FUNCTION_BLOCK Starting IMPLEMENTS ITF_PackMLState
VAR
	_MyContext : REFERENCE TO SomeMachine;
END_VAR

METHOD CyclicLogic : BOOL
VAR_INPUT
END_VAR
END_METHOD

{warning 'add method implementation '}
METHOD EStop : BOOL
END_METHOD

{warning 'add method implementation '}
METHOD Reset : BOOL
END_METHOD

METHOD SetContext : BOOL
VAR_INPUT
	context	: REFERENCE TO SomeMachine;
END_VAR
_MyContext REF= context;
END_METHOD

{warning 'add method implementation '}
METHOD Start : BOOL
END_METHOD

{warning 'add method implementation '}
METHOD Stop : BOOL
END_METHOD

END_FUNCTION_BLOCK

(* stored: Version 1.1.0.1, ProductVersion 3.1.4024.12
   POU Starting: Id {624bebe4-67c6-44f5-beab-72635c155632}, SpecialFunc None
   Method CyclicLogic: Id {3254b99f-1dc0-4979-8be0-c95b78edab85}
   Method EStop: Id {6cc05f29-5f9f-4b95-af67-3fa6d6332d92}
   Method Reset: Id {78ca631f-4d7b-4599-bf61-fb545cd859b2}
   Method SetContext: Id {908bd32b-87e0-4973-b00d-138bba61c875}
   Method Start: Id {e09d86fc-5ae2-4b3a-b400-588448b4ef81}
   Method Stop: Id {27297469-e38c-448f-97df-f229cd1d7c5e} *)
